FUNCTION_BLOCK Attribute_ID (* Input service interface function block for VT object attribute indication and response data *)
  (* Description: Copyright (c) 2026 HR Agrartechnik GmbH This program and the accompanying materials are made available under the terms of the Eclipse Public License 2.0 which is available at https://www.eclipse.org/legal/epl-2.0/ SPDX-License-Identifier: EPL-2.0 *)
  (* Version 1.0, 2026-09-15, Franz Höpfinger, HR Agrartechnik GmbH, Initial implementation of Attribute_ID input service interface *)
  PACKAGE isobus::UT::I;
  IMPORT isobus::UT::Q::const::IDs::ID_NULL;
  (* Documentation:
  Attribute_ID Input Service Interface
   Input service interface function block for receiving asynchronous VT object attribute values. Serves as an input interface for VT attribute indications (IND) and confirmations (CNF).
  *)
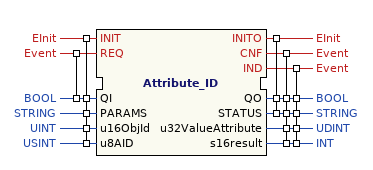
  EVENT_INPUT
    INIT : EInit WITH QI, PARAMS, u16ObjId, u8AID; (* Service Initialization *)
    REQ WITH QI; (* Service Request *)
  END_EVENT
  EVENT_OUTPUT
    INITO : EInit WITH QO, STATUS; (* Initialization Confirm *)
    CNF WITH QO, STATUS, u32ValueAttribute, s16result; (* Confirmation of Requested Service *)
    IND WITH QO, STATUS, u32ValueAttribute, s16result; (* Indication from Resource *)
  END_EVENT
  VAR_INPUT
    QI : BOOL; (* Event Input Qualifier *)
    PARAMS : STRING; (* Service Parameters *)
    u16ObjId : UINT := ID_NULL; (* Object ID *)
    u8AID : USINT; (* Attribute ID of the object *)
  END_VAR
  VAR_OUTPUT
    QO : BOOL; (* Event Output Qualifier *)
    STATUS : STRING; (* Service Status *)
    u32ValueAttribute : UDINT; (* value for attribute *)
    s16result : INT; (* retval see description *)
  END_VAR
END_FUNCTION_BLOCK
